// TIA Portal V17 export
// export: Created 2023-04-06T14:59:51.4519566Z, ExportSetting None, DisplayName Totally Integrated Automation Portal, DisplayVersion V17 Update 4, DisplayName TIA Portal Openness, DisplayVersion V17 Update 4, DisplayName TIA Portal Version Control Interface, DisplayVersion V17, DisplayName STEP 7 Professional, DisplayVersion V17 Update 4, DisplayName STEP 7 Safety, DisplayVersion V17, DisplayName WinCC Advanced / Unified PC, DisplayVersion V17 Update 4
DATA_BLOCK "SETTINGS"   // DB26
{ S7_Optimized_Access := 'FALSE' }
// stored: AutoNumber false
   VAR RETAIN
      PT_104 : Struct   // GAS SUCTION PRESSURE
         RANGE_L : Real := -1.0;
         RANGE_H : Real := 40.0;
         SP_LL : Real := -101.0;
         SP_L : Real := 0.0;
         SP_H : Real := 0.8;
         SP_HH : Real := 140.0;
      END_STRUCT;
      TT_107_1 : Struct   // GAS SUCTION TEMPERATURE
         RANGE_L : Real := -50.0;
         RANGE_H : Real := 120.0;
         SP_LL : Real := -150.0;
         SP_L : Real := 5.0;
         SP_H : Real := 50.0;
         SP_HH : Real := 220.0;
      END_STRUCT;
      PT_124 : Struct   // GAS DISCHARGE PRESSURE
         RANGE_L : Real := -1.0;
         RANGE_H : Real := 40.0;
         SP_LL : Real := -101.0;
         SP_L : Real := -101.0;
         SP_H : Real := 22.4;
         SP_HH : Real := 140.0;
      END_STRUCT;
      PDT_120 : Struct   // DIFFERENTIAL PRESSURE GAS-OIL SEPARATOR
         RANGE_L : Real := 0.0;
         RANGE_H : Real := 1000.0;
         SP_LL : Real := -100.0;
         SP_L : Real := -100.0;
         SP_H : Real := 250.0;
         SP_HH : Real := 1100.0;
      END_STRUCT;
      PDT_121 : Struct   // 1st STAGE FILTER DIFFERENTIAL PRESSURE
         RANGE_L : Real := 0.0;
         RANGE_H : Real := 1000.0;
         SP_LL : Real := -100.0;
         SP_L : Real := -100.0;
         SP_H : Real := 300.0;
         SP_HH : Real := 1100.0;
      END_STRUCT;
      PDT_122 : Struct   // 2nd STAGE FILTER DIFFERENTIAL PRESSURE
         RANGE_L : Real := 0.0;
         RANGE_H : Real := 1000.0;
         SP_LL : Real := -100.0;
         SP_L : Real := -100.0;
         SP_H : Real := 300.0;
         SP_HH : Real := 1100.0;
      END_STRUCT;
      PDT_123 : Struct   // 3rd STAGE FILTER DIFFERENTIAL PRESSURE
         RANGE_L : Real := 0.0;
         RANGE_H : Real := 1000.0;
         SP_LL : Real := -100.0;
         SP_L : Real := -100.0;
         SP_H : Real := 300.0;
         SP_HH : Real := 1100.0;
      END_STRUCT;
      PDT_124 : Struct   // 4th STAGE FILTER DIFFERENTIAL PRESSURE
         RANGE_L : Real := 0.0;
         RANGE_H : Real := 1000.0;
         SP_LL : Real := -100.0;
         SP_L : Real := -100.0;
         SP_H : Real := 300.0;
         SP_HH : Real := 1100.0;
      END_STRUCT;
      GT_123_3 : Struct   // RECYCLE VALVE POSITION FEEDBACK
         RANGE_L : Real := 0.0;
         RANGE_H : Real := 100.0;
         SP_LL : Real := -100.0;
         SP_L : Real := -100.0;
         SP_H : Real := 200.0;
         SP_HH : Real := 200.0;
      END_STRUCT;
      PDT_206 : Struct   // PRIMARY OIL FILTER DIFFERENTIAL PRESSURE
         RANGE_L : Real := 0.0;
         RANGE_H : Real := 1000.0;
         SP_LL : Real := -100.0;
         SP_L : Real := -100.0;
         SP_H : Real := 500.0;
         SP_HH : Real := 1100.0;
      END_STRUCT;
      GT_450_3 : Struct   // WATER CONTROL VALVE POSITION FEEDBACK
         RANGE_L : Real := 0.0;
         RANGE_H : Real := 100.0;
         SP_LL : Real := -100.0;
         SP_L : Real := -100.0;
         SP_H : Real := 200.0;
         SP_HH : Real := 200.0;
      END_STRUCT;
      GT_440 : Struct   // WATER CONTROL VALVE POSITION FEEDBACK
         RANGE_L : Real := 0.0;
         RANGE_H : Real := 100.0;
         SP_LL : Real := -100.0;
         SP_L : Real := -100.0;
         SP_H : Real := 200.0;
         SP_HH : Real := 200.0;
      END_STRUCT;
      GT_168 : Struct   // SLIDE VALVE POSITION FEEDBACK
         RANGE_L : Real := 0.0;
         RANGE_H : Real := 100.0;
         SP_LL : Real := -100.0;
         SP_L : Real := 35.0;
         SP_H : Real := 200.0;
         SP_HH : Real := 200.0;
      END_STRUCT;
      TT_125 : Struct   // GAS TEMPERATURE DOWNSTREAM GAS COOLER
         RANGE_L : Real := -50.0;
         RANGE_H : Real := 120.0;
         SP_LL : Real := -150.0;
         SP_L : Real := 15.0;
         SP_H : Real := 50.0;
         SP_HH : Real := 220.0;
      END_STRUCT;
      KF_401 : Struct   // SET SLIDE POSITION
         RANGE_L : Real := 0.0;
         RANGE_H : Real := 100.0;
         SP_LL : Real := -100.0;
         SP_L : Real := -100.0;
         SP_H : Real := 200.0;
         SP_HH : Real := 200.0;
      END_STRUCT;
      KF_408 : Struct   // SET RECYCLE VALVE POSITION
         RANGE_L : Real := 0.0;
         RANGE_H : Real := 100.0;
         SP_LL : Real := -100.0;
         SP_L : Real := -100.0;
         SP_H : Real := 200.0;
         SP_HH : Real := 200.0;
      END_STRUCT;
      PGP_202 : Struct   // CALCULATED OIL - GAS PRESSURE RATIO (PT124 / PT105)
         RANGE_L : Real := 0.5;
         RANGE_H : Real := 25.0;
         SP_LL : Real := 1.5;
         SP_L : Real := 1.5;
         SP_H : Real := 20.0;
         SP_HH : Real := 23.0;
      END_STRUCT;
      PDP_203 : Struct   // CALCULATED COMPRESSOR DIFFERENTIAL PRESSURE (PT124 - PT105)
         RANGE_L : Real := 0.5;
         RANGE_H : Real := 25.0;
         SP_LL : Real := 3.0;
         SP_L : Real := 3.5;
         SP_H : Real := 125.0;
         SP_HH : Real := 125.0;
      END_STRUCT;
      PT_105 : Struct   // GAS SUCTION PRESSURE
         RANGE_L : Real := -1.0;
         RANGE_H : Real := 40.0;
         SP_LL : Real := 0.3;
         SP_L : Real := -101.0;
         SP_H : Real := 140.0;
         SP_HH : Real := 1.2;
      END_STRUCT;
      PT_113 : Struct   // GAS DISCHARGE PRESSURE
         RANGE_L : Real := -1.0;
         RANGE_H : Real := 40.0;
         SP_LL : Real := -101.0;
         SP_L : Real := -101.0;
         SP_H : Real := 22.7;
         SP_HH : Real := 23.0;
      END_STRUCT;
      TT_114 : Struct   // GAS DISCHARGE TEMPERATURE
         RANGE_L : Real := -50.0;
         RANGE_H : Real := 120.0;
         SP_LL : Real := -150.0;
         SP_L : Real := -150.0;
         SP_H : Real := 110.0;
         SP_HH : Real := 115.0;
      END_STRUCT;
      TT_128 : Struct   // GAS TEMPERATURE DOWNSTREAM GAS COOLER
         RANGE_L : Real := -50.0;
         RANGE_H : Real := 120.0;
         SP_LL : Real := -150.0;
         SP_L : Real := -150.0;
         SP_H : Real := 220.0;
         SP_HH : Real := 60.0;
      END_STRUCT;
      TT_208 : Struct   // LUBE OIL TEMPERATURE
         RANGE_L : Real := -50.0;
         RANGE_H : Real := 120.0;
         SP_LL : Real := -150.0;
         SP_L : Real := 25.0;
         SP_H : Real := 65.0;
         SP_HH : Real := 70.0;
      END_STRUCT;
      PT_501 : Struct   // INSTRUMENT AIR PRESSURE
         RANGE_L : Real := -1.0;
         RANGE_H : Real := 40.0;
         SP_LL : Real := 4.5;
         SP_L : Real := -101.0;
         SP_H : Real := 140.0;
         SP_HH : Real := 26.0;
      END_STRUCT;
      VT_111_13 : Struct   // COMPRESSOR HOUSING VIBRATION
         RANGE_L : Real := 0.0;
         RANGE_H : Real := 25.4;
         SP_LL : Real := -100.0;
         SP_L : Real := -100.0;
         SP_H : Real := 4.5;
         SP_HH : Real := 6.0;
      END_STRUCT;
      VT_112_13 : Struct   // MAIN MOTOR BEARING DE VIBRATION
         RANGE_L : Real := 0.0;
         RANGE_H : Real := 25.4;
         SP_LL : Real := -100.0;
         SP_L : Real := -100.0;
         SP_H : Real := 4.5;
         SP_HH : Real := 6.0;
      END_STRUCT;
      VT_112_14 : Struct   // MAIN MOTOR BEARING NDE VIBRATION
         RANGE_L : Real := 0.0;
         RANGE_H : Real := 25.4;
         SP_LL : Real := -100.0;
         SP_L : Real := -100.0;
         SP_H : Real := 4.5;
         SP_HH : Real := 6.0;
      END_STRUCT;
      TE_112_5_I : Struct   // MAIN MOTOR WINDING TEMPERATURE U
         RANGE_L : Real := 0.0;
         RANGE_H : Real := 200.0;
         SP_LL : Real := -100.0;
         SP_L : Real := -100.0;
         SP_H : Real := 130.0;
         SP_HH : Real := 145.0;
      END_STRUCT;
      TE_112_6_I : Struct   // MAIN MOTOR WINDING TEMPERATURE V
         RANGE_L : Real := 0.0;
         RANGE_H : Real := 200.0;
         SP_LL : Real := -100.0;
         SP_L : Real := -100.0;
         SP_H : Real := 130.0;
         SP_HH : Real := 145.0;
      END_STRUCT;
      TE_112_7_I : Struct   // MAIN MOTOR WINDING TEMPERATURE W
         RANGE_L : Real := 0.0;
         RANGE_H : Real := 200.0;
         SP_LL : Real := -100.0;
         SP_L : Real := -100.0;
         SP_H : Real := 130.0;
         SP_HH : Real := 145.0;
      END_STRUCT;
   END_VAR
BEGIN
END_DATA_BLOCK
